(* IEC 61131-3 sources: industrial-controls-learning-lab/examples/structured-text, 4 files *)

(* ---- E_EquipmentState.st ---- *)
TYPE E_EquipmentState :
(
    IDLE := 0,
    READY := 10,
    RUNNING := 20,
    STOPPING := 30,
    FAULT := 900,
    RESETTING := 910
);
END_TYPE

(* ---- E_MotionBlockReason.st ---- *)
TYPE E_MotionBlockReason :
(
    NONE := 0,
    EMERGENCY_STOP_ACTIVE := 10,
    GUARD_OPEN := 20,
    NETWORK_UNHEALTHY := 30,
    DRIVE_FAULT := 40,
    EXTERNAL_PERMISSION_MISSING := 50
);
END_TYPE

(* ---- FB_EquipmentStateMachine.st ---- *)
FUNCTION_BLOCK FB_EquipmentStateMachine
VAR_INPUT
    bEnableRequest : BOOL;
    bStartEdge : BOOL;
    bStopRequest : BOOL;
    bStopComplete : BOOL;
    bMotionAllowed : BOOL;
    bFaultActive : BOOL;
    bResetEdge : BOOL;
END_VAR
VAR_OUTPUT
    eState : E_EquipmentState := E_EquipmentState.IDLE;
    bRunCommand : BOOL;
END_VAR

bRunCommand := FALSE;

IF bFaultActive AND (eState <> E_EquipmentState.FAULT) THEN
    eState := E_EquipmentState.FAULT;
END_IF

CASE eState OF
    E_EquipmentState.IDLE:
        IF bEnableRequest AND bMotionAllowed THEN
            eState := E_EquipmentState.READY;
        END_IF

    E_EquipmentState.READY:
        IF bStartEdge AND bMotionAllowed THEN
            eState := E_EquipmentState.RUNNING;
        END_IF

    E_EquipmentState.RUNNING:
        bRunCommand := bMotionAllowed;
        IF (NOT bMotionAllowed) OR bFaultActive THEN
            eState := E_EquipmentState.FAULT;
        ELSIF bStopRequest THEN
            eState := E_EquipmentState.STOPPING;
        END_IF

    E_EquipmentState.STOPPING:
        IF bStopComplete THEN
            eState := E_EquipmentState.READY;
        END_IF

    E_EquipmentState.FAULT:
        IF bResetEdge AND (NOT bFaultActive) THEN
            eState := E_EquipmentState.RESETTING;
        END_IF

    E_EquipmentState.RESETTING:
        eState := E_EquipmentState.IDLE;
END_CASE

(* ---- FB_MotionPermission.st ---- *)
FUNCTION_BLOCK FB_MotionPermission
VAR_INPUT
    bEmergencyStopReleased : BOOL;
    bGuardClosed : BOOL;
    bNetworkHealthy : BOOL;
    bDriveFault : BOOL;
    bExternalPermission : BOOL;
END_VAR
VAR_OUTPUT
    bMotionAllowed : BOOL;
    eBlockReason : E_MotionBlockReason;
END_VAR

bMotionAllowed := FALSE;
eBlockReason := E_MotionBlockReason.NONE;

IF NOT bEmergencyStopReleased THEN
    eBlockReason := E_MotionBlockReason.EMERGENCY_STOP_ACTIVE;
ELSIF NOT bGuardClosed THEN
    eBlockReason := E_MotionBlockReason.GUARD_OPEN;
ELSIF NOT bNetworkHealthy THEN
    eBlockReason := E_MotionBlockReason.NETWORK_UNHEALTHY;
ELSIF bDriveFault THEN
    eBlockReason := E_MotionBlockReason.DRIVE_FAULT;
ELSIF NOT bExternalPermission THEN
    eBlockReason := E_MotionBlockReason.EXTERNAL_PERMISSION_MISSING;
ELSE
    bMotionAllowed := TRUE;
END_IF
